// TIA Portal V20 export
TYPE "HMIAxisCtrl_typeInternal"
TITLE = HMIAxisCtrl_typeInternal
// Support: tech.team.motioncontrol@siemens.com 
// Fax: +49 (0) 9131/98-1297
   STRUCT
      mode : Int := -1;   // Internal mode identifier; 1: Jog ; 2: Move; 3: Pos; 4: Homing; 5: Brake
      absoluteSelected : Bool;   // TRUE: Absolute positioning; FALSE: Relative positioning
      isPosRelative : Bool;   // TRUE: Show controls related to relative positioning
      isPosAbsoluteWithModulo : Bool;   // TRUE: Show controls related to absolute positioning (with modulo)
      isPosAbsoluteWithoutModulo : Bool;   // TRUE: Show controls related to absolute positioning (without modulo)
      isAxisWithIncrementalEncoder : Bool;   // TRUE: Show controls related to axis with incremental encoder
      isAxisWithAbsoluteEncoder : Bool;   // TRUE: Show controls related to axis with absolute encoder
      isNotExternalEncoder : Bool;   // TRUE: Show controls related to homing functionality of axis (not external encoder)
      velocity : LReal := -1.0;   // Internal variable for velocity input
      position : LReal := 0.0;   // Internal variable for position input
      acceleration : LReal := -1.0;   // Internal variable for acceleration input
      deceleration : LReal := -1.0;   // Internal variable for deceleration input
      jerk : LReal := -1.0;   // Internal variable for jerk input
   END_STRUCT;
END_TYPE
